Omron CX-Programmer project NuevoProyecto (CX-Programmer 9.75)

# PLC Git_test: CJ2M CPU11

## Program NuevoPrograma1 (cyclic task 0)

### Section Sección1

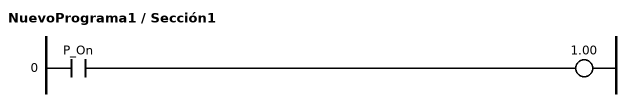
; rung 0
LD P_On
OUT 1.00

### Section SeccionGeras

### Section END
; rung 0
END(001)